Omron Sysmac Studio project YukselenDusenKenar (Sysmac Studio 1.65.0.64007, StandardProject)

# Controller new_Controller_0: NX1P2-1040DT1 version 1.69
Task PrimaryTask (priority 4, period or condition 2000): Program0

VAR_GLOBAL
    IN_Start_Button : BOOL;
    IN_Stop_Button : BOOL;
    OUT_KonveyorMotor : BOOL;
    IN_OptikSensor : BOOL;
    E_KoliSayma : INT;
    BIO_Input_Bit_00 : BOOL;  (* at BuiltInIO://cpu/#0/Input_Bit_00 *)
    BIO_Input_Bit_01 : BOOL;  (* at BuiltInIO://cpu/#0/Input_Bit_01 *)
    BIO_Input_Bit_02 : BOOL;  (* at BuiltInIO://cpu/#0/Input_Bit_02 *)
    BIO_Output_Bit_00 : BOOL;  (* at BuiltInIO://cpu/#0/Output_Bit_00 *)
END_VAR

PROGRAM Program0
VAR
    DusenKenarFBR : F_TRIG;
END_VAR
VAR_EXTERNAL
    IN_Start_Button : BOOL;
    IN_Stop_Button : BOOL;
    OUT_KonveyorMotor : BOOL;
    IN_OptikSensor : BOOL;
    E_KoliSayma : INT;
    BIO_Input_Bit_00 : BOOL;
    BIO_Input_Bit_01 : BOOL;
    BIO_Input_Bit_02 : BOOL;
    BIO_Output_Bit_00 : BOOL;
END_VAR
VAR
    _e1 : R_TRIG;
    _e2 : F_TRIG;
    _e3 : R_TRIG;
END_VAR

(* Section InOut: ladder, written here as Structured Text *)

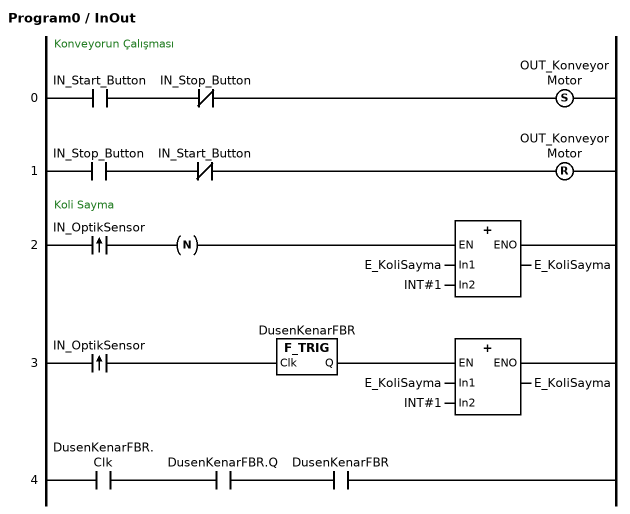
(* Rung 0: Konveyorun Çalışması *)
IF IN_Start_Button AND NOT IN_Stop_Button THEN OUT_KonveyorMotor := TRUE; END_IF;
(* Rung 1 *)
IF IN_Stop_Button AND NOT IN_Start_Button THEN OUT_KonveyorMotor := FALSE; END_IF;
(* Rung 2: Koli Sayma *)
_e1(CLK := IN_OptikSensor);
_e2(CLK := _e1.Q);
IF _e2.Q THEN E_KoliSayma := E_KoliSayma + INT#1; END_IF;
(* Rung 3 *)
_e3(CLK := IN_OptikSensor);
DusenKenarFBR(Clk := _e3.Q);
IF DusenKenarFBR.Q THEN E_KoliSayma := E_KoliSayma + INT#1; END_IF;
(* Rung 4 *)
(* drawn but driving nothing: DusenKenarFBR.Clk, DusenKenarFBR.Q, DusenKenarFBR *)

(* Section Konveyor_KoliSayma: ladder, written here as Structured Text *)

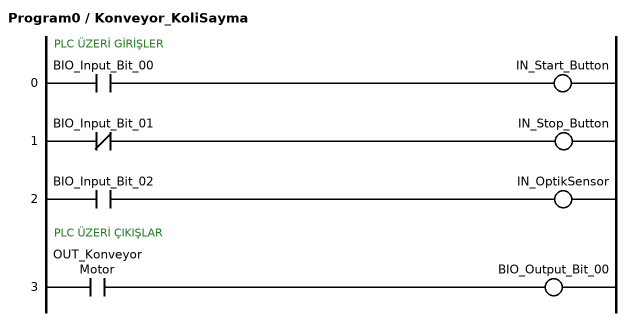
(* Rung 0: PLC ÜZERİ GİRİŞLER *)
IN_Start_Button := BIO_Input_Bit_00;
(* Rung 1 *)
IN_Stop_Button := NOT BIO_Input_Bit_01;
(* Rung 2 *)
IN_OptikSensor := BIO_Input_Bit_02;
(* Rung 3: PLC ÜZERİ ÇIKIŞLAR *)
BIO_Output_Bit_00 := OUT_KonveyorMotor;
END_PROGRAM